TYPE ST_Station_2 :
STRUCT
	
	Mov1				: BOOL;		
	Mov2				: BOOL;	
	Mov3				: BOOL;		
	
END_STRUCT
END_TYPE

(* stored: Version 1.1.0.1, ProductVersion 3.1.4024.13
   DUT ST_Station_2: Id {5e9725c2-a62b-4a6e-833a-62a48f17fc9a} *)
